TYPE ST_Alarm :
STRUCT
	dtDateTime		: DATE_AND_TIME;
	sName			: STRING;
	nCategory		: DINT;
	nCode			: DINT;
	sMessage		: STRING(255);
END_STRUCT
END_TYPE

(* stored: Version 1.1.0.1, ProductVersion 3.1.4024.12
   DUT ST_Alarm: Id {1f186126-39b4-4c54-a3b6-a9934edd8fe5} *)
